FUNCTION_BLOCK ColorMap (* Basic Function Block Type *)
  (* Standard: 61499-2 *)
  (* Version 0.0, 22/06/2022, Lernfabrik, WBK hackaton, Template *)
  PACKAGE Main;
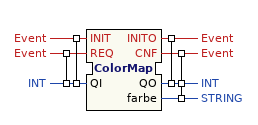
  EVENT_INPUT
    INIT WITH QI; (* Initialization Request *)
    REQ WITH QI; (* Normal Execution Request *)
  END_EVENT
  EVENT_OUTPUT
    INITO WITH QO; (* Initialization Confirm *)
    CNF WITH QO, farbe; (* Execution Confirmation *)
  END_EVENT
  VAR_INPUT
    QI : INT; (* Input event qualifier *)
  END_VAR
  VAR_OUTPUT
    QO : INT; (* Output event qualifier *)
    farbe : STRING; (* olo *)
  END_VAR
  VAR
    Minimum : INT;
    SAMPLECOUNT : INT := 0;
  END_VAR
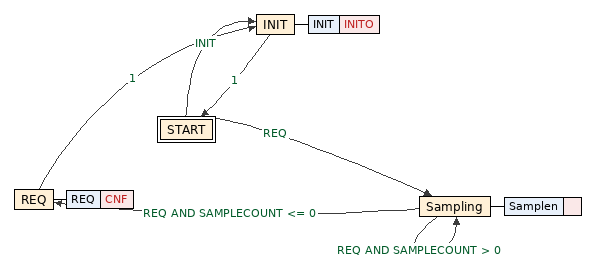
  EC_STATES
    START; (* Initial State *)
    INIT : INIT -> INITO; (* Initialization *)
    REQ : REQ -> CNF; (* Normal execution *)
    Sampling : Samplen;
  END_STATES
  EC_TRANSITIONS
    START TO INIT := INIT;
    INIT TO START := 1;
    START TO Sampling := REQ;
    Sampling TO Sampling := REQ AND SAMPLECOUNT > 0;
    Sampling TO REQ := REQ AND SAMPLECOUNT <= 0;
    REQ TO INIT := 1;
  END_TRANSITIONS
  ALGORITHM INIT IN ST: (* Initialization algorithm *)
Minimum := 32000;
QO := Minimum;
farbe := 'NONE';
  END_ALGORITHM
  ALGORITHM REQ IN ST: (* Normally executed algorithm *)
farbe := 'NONE';

IF  Minimum <20300
THEN
farbe := 'WHITE';
END_IF;

IF  Minimum > 20850 AND Minimum <21450
THEN
farbe := 'RED';
END_IF;

IF  Minimum > 26650 AND Minimum < 27300
	THEN
	farbe := 'BLUE';
END_IF;
  END_ALGORITHM
  ALGORITHM Samplen IN ST:
IF QI < 27400 THEN
	(* Starte Sampling, weil eine Farbe erkannt wurde *)
	SAMPLECOUNT := 1;
END_IF;

IF SAMPLECOUNT > 0 AND QI > 27400 THEN
	(* Warte, ob nur ein Ausreißer war, sonst stoppen *)
	SAMPLECOUNT := SAMPLECOUNT - 1;
ELSIF SAMPLECOUNT > 0 AND QI < 27400 THEN
	(* Reset: Doch weiter samplen, war wohl nur ein Ausreißer *)
	SAMPLECOUNT := 1;
END_IF;

IF SAMPLECOUNT > 0 AND QI < Minimum THEN
	Minimum := QI;
END_IF;

QO := Minimum;
;
  END_ALGORITHM
END_FUNCTION_BLOCK
